FUNCTION_BLOCK FanControl
VAR_IN_OUT
	Parameters:GreenMasterBaseParameters;
END_VAR
VAR_INPUT
	EN: BOOL;
	ControlMode: FanControlTypes;
	ControlParameters: ControllerParameters;
	Pressure: LREAL;
	PressureError: BOOL;
	Flow: LREAL;
	FlowError: BOOL;
	MasterPV: LREAL;
	FanAlarm: BOOL;
	MinSpeed: LREAL := 0;
	MaxSpeed: LREAL := 1;
	Override: BOOL;
	OverrideCV: LREAL;
	ExtendedOperation: BOOL;
	PostVentilationTime: LTIME := LTIME#2M;
	Fire: BOOL;
	Damper: BOOL := TRUE;
END_VAR
VAR_OUTPUT
	ENO: BOOL;
	CV: LREAL;
	PV: LREAL;
	FanRunning: BOOL;
	Recirculation: BOOL;
END_VAR
VAR
	Fan: Fan;
	Ramp: Ramp;
	PiController: PidController;
	StartDelay: TON;
	SPC: Interpolate;
	SupplyAirControl: SupplyAirControl;
	MAX_FB_0: MAX_FB;
	MIN_FB_0: MIN_FB;
	TON_0: TON;
	ControlP: LREAL;
	ControlI: TIME;
	ControlSP: LREAL;
	PostVentilation: PostVentilation;
END_VAR
VAR // added by the converter: edge detectors and wires of the graphical bodies
    _w1, _w2, _w3, _w4, _w5, _w7, _w8, _w9 : ANY;
    _w6 : BOOL;
END_VAR


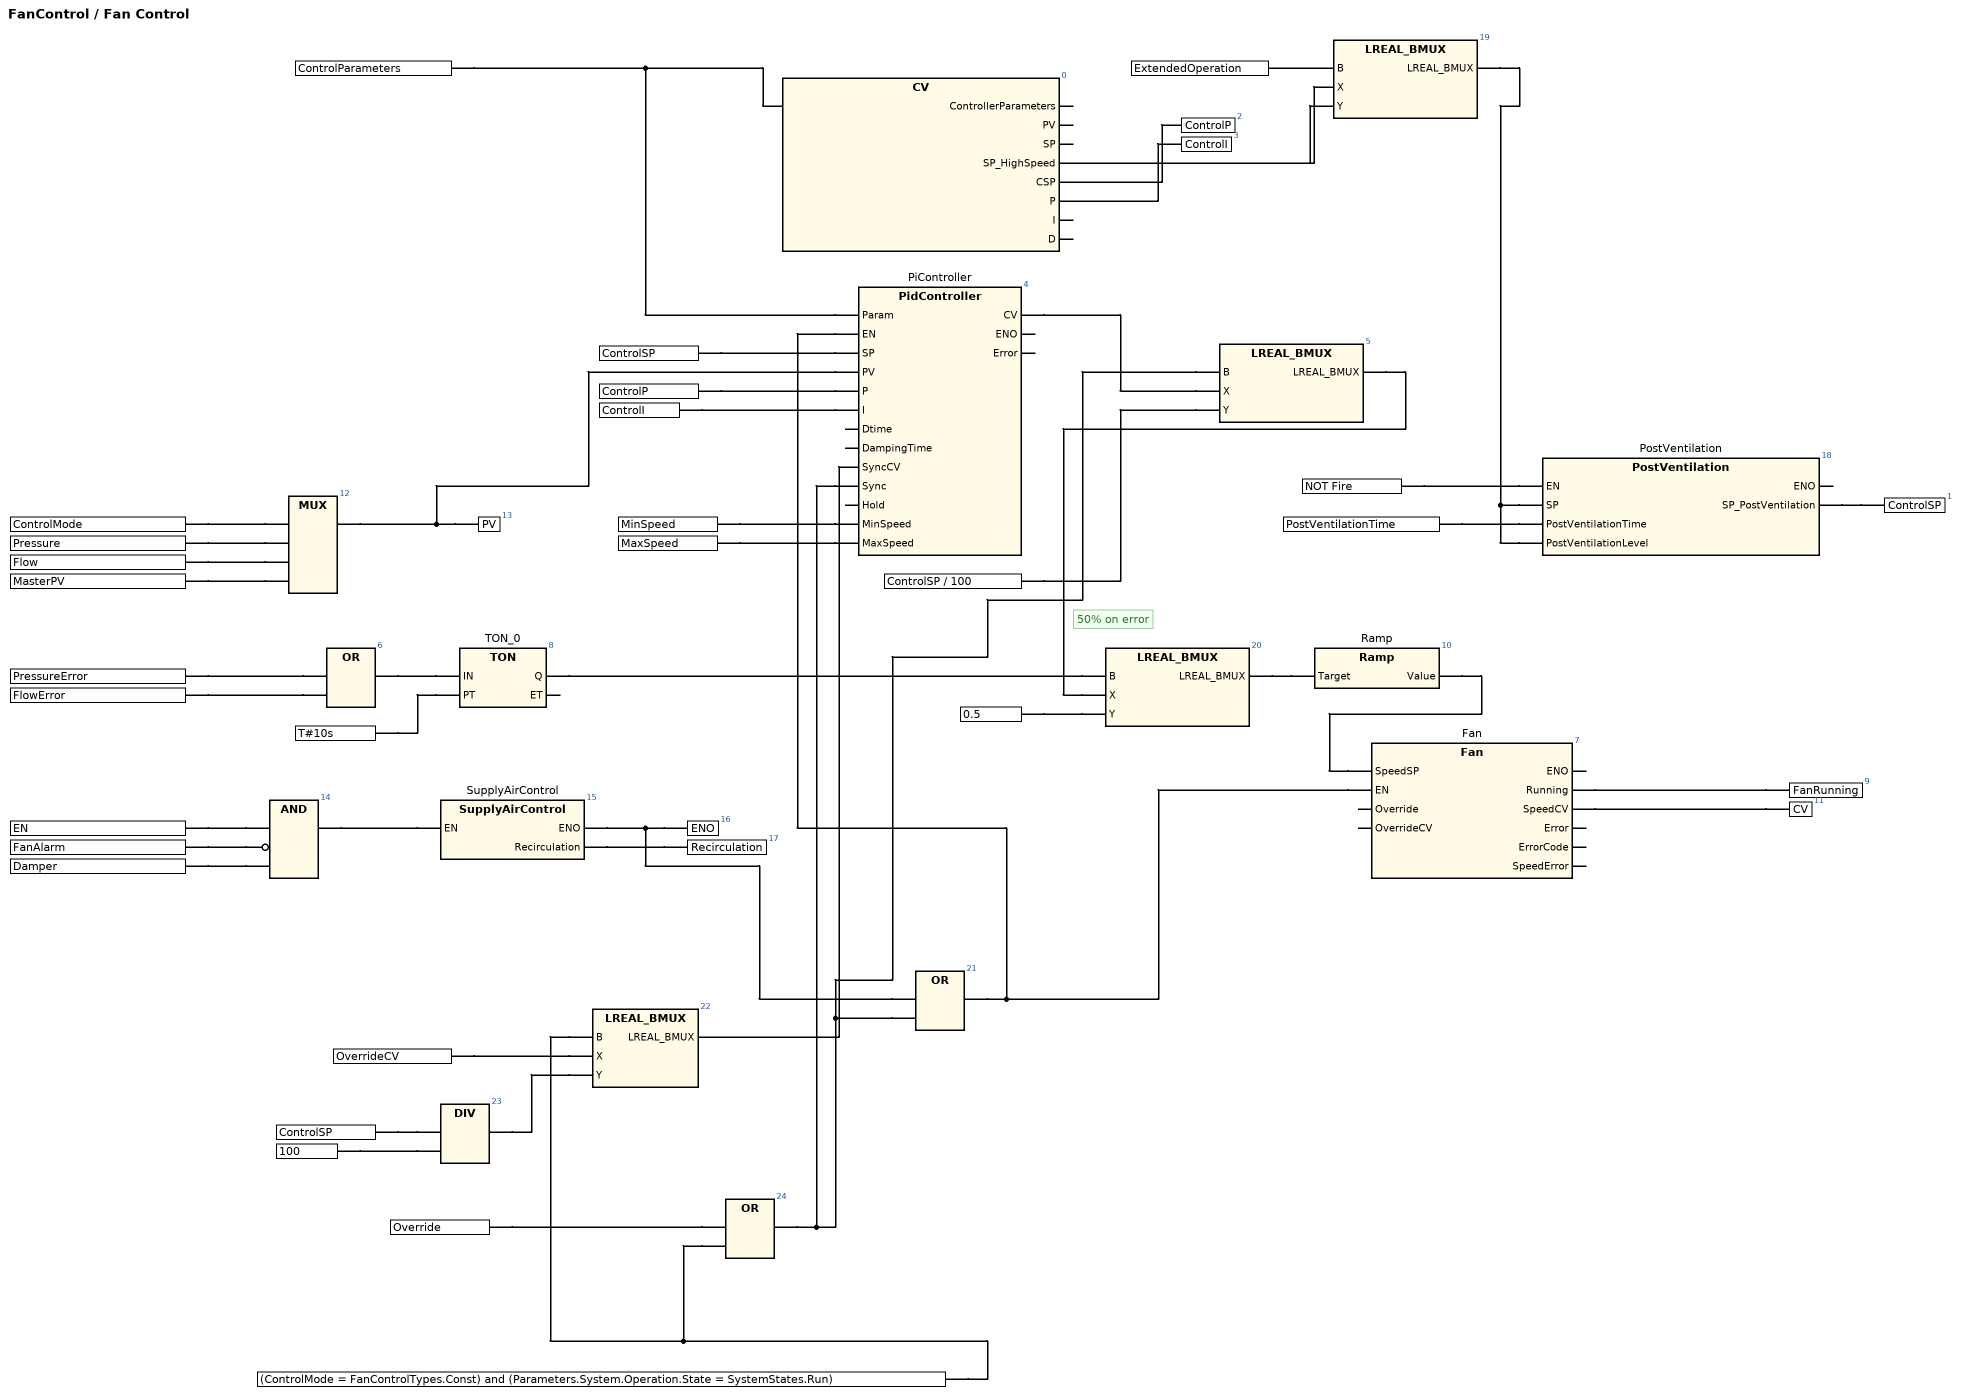
// PAGE Fan Control
ControlSP := PostVentilation.SP_PostVentilation;
ControlP := ControlParameters.CSP;
ControlI := ControlParameters.P;
PiController(
    Param := ControlParameters,
    EN := _w1,
    SP := ControlSP,
    PV := _w2,
    P := ControlP,
    I := ControlI,
    SyncCV := _w3,
    Sync := _w4,
    MinSpeed := MinSpeed,
    MaxSpeed := MaxSpeed); // PidController
_w5 := LREAL_BMUX(B := _w4, X := PiController.CV, Y := ControlSP / 100);
_w6 := PressureError OR FlowError;
Fan(SpeedSP := Ramp.Value, EN := _w1);
TON_0(IN := _w6, PT := T#10s); // TON
FanRunning := Fan.Running;
Ramp(Target := _w7);
CV := Fan.SpeedCV;
_w2 := MUX(ControlMode, Pressure, Flow, MasterPV);
PV := _w2;
SupplyAirControl(EN := EN AND NOT FanAlarm AND Damper);
ENO := SupplyAirControl.ENO;
Recirculation := SupplyAirControl.Recirculation;
PostVentilation(
    EN := NOT Fire,
    SP := _w8,
    PostVentilationTime := PostVentilationTime,
    PostVentilationLevel := _w8);
_w8 := LREAL_BMUX(B := ExtendedOperation, X := ControlParameters.SP_HighSpeed, Y := ControlParameters.SP_HighSpeed);
// 50% on error
_w7 := LREAL_BMUX(B := TON_0.Q, X := _w5, Y := 0.5);
_w1 := SupplyAirControl.ENO OR _w4;
_w3 := LREAL_BMUX(B := (ControlMode = FanControlTypes.Const) and (Parameters.System.Operation.State = SystemStates.Run), X := OverrideCV, Y := _w9);
_w9 := ControlSP / 100;
_w4 := Override OR ((ControlMode = FanControlTypes.Const) and (Parameters.System.Operation.State = SystemStates.Run));

END_FUNCTION_BLOCK

(* stored: Version 1.1.0.1, ProductVersion 3.1.4024.6
   POU FanControl: Id {62ee3baf-57b6-4b81-850b-e42bf6d60791}, SpecialFunc None *)
